TEXTLIST TL_E_CTRL_STATION
  0 = 'STATION_CTRL_NULL'
  1 = 'STATION_INIT'
  10 = 'STATION_DISABLE'
  11 = 'STATION_ENABLE'
  20 = 'STATION_MOVER_ENTER'
  21 = 'STATION_MOVER_ENTER_RETRY'
  22 = 'STATION_MOVER_SEND'
  30 = 'STATION_PROCESS_START'
  31 = 'STATION_PROCESS_DONE'
  50 = 'STATION_MOVER_OUT'
  51 = 'STATION_MOVER_OUT_RETRY'
  60 = 'STATION_MOVER_GONE'
   = ''
END_TEXTLIST

(* stored: Version 1.1.0.1
   TextList TL_E_CTRL_STATION: Id {a17b364b-ec6a-4a27-a9df-a84e89340f10} *)
